TYPE U_DEVICE_COM_CACHE :
UNION
	Text				:	STRING(PARAM.DEVICE_COM_MAX_CACHE-1);
	Bytes				:	ARRAY[PARAM.DEVICE_COM_MIN_CACHE..PARAM.DEVICE_COM_MAX_CACHE] OF BYTE;	
END_UNION
END_TYPE

(* stored: Version 1.1.0.1, ProductVersion 3.1.4024.13
   DUT U_DEVICE_COM_CACHE: Id {74595ac0-be83-4795-8f43-5c4bd6cf16e5} *)
